FUNCTION_BLOCK FB_Kuka_KRC2
VAR_INPUT
END_VAR
VAR_OUTPUT
END_VAR
VAR
END_VAR

END_FUNCTION_BLOCK

(* stored: Version 1.1.0.1, ProductVersion 3.1.4024.9
   POU FB_Kuka_KRC2: Id {a64a119b-0352-4618-9447-2528436fe8a6}, SpecialFunc None *)
